// TIA Portal project "lab4" (V15)
// generatory

(* hardware
DEVICE "S7-1200 station_1"  S7-1200 Station
   slot 0: "Rack_0"  S7-1200 Rack  Rack  V1.0
   slot 1: "PLC_1"  CPU 1214C DC/DC/DC  6ES7 214-1AG40-0XB0  V4.2
      slot 3: "AQ 1x12BIT_1"  AQ1 signal board  6ES7 232-4HA30-0XB0  V1.0
   slot 101: "CM 1243-5"  CM 1243-5  6GK7 243-5DX30-0XE0  V1.3
   slot 102: "CM 1241 (RS485)_1"  CM 1241 (RS485)  6ES7 241-1CH30-0XB0  V1.0
*)

// ===== PLC "PLC_1"  CPU 1214C DC/DC/DC =====

VAR_GLOBAL   // PLC tag table "Default tag table"
   "start1" AT %I0.0 : Bool;
   "sprzezenie1" AT %M0.0 : Bool;
   "wyjscie1" AT %Q0.0 : Bool;
   "start2" AT %I0.1 : Bool;
   "sprzezenie2" AT %M0.2 : Bool;
   "WY_1" AT %Q0.2 : Bool;
   "start3" AT %I0.4 : Bool;
   "sprzezenie3" AT %M0.3 : Bool;
   "WY" AT %Q0.3 : Bool;
   "start5" AT %I0.5 : Bool;
   "sprzezenie4" AT %M0.5 : Bool;
   "wyjscie5" AT %Q0.5 : Bool;
   "szpikaZbocze" AT %M1.0 : Bool;
END_VAR

// folder: System blocks/Program resources

DATA_BLOCK "T1"   // DB1
{ S7_Optimized_Access := 'TRUE' }
AUTHOR : Simatic
FAMILY : IEC
NAME : IEC_TMR
VERSION : 1.0
// stored: InstanceOfName IEC_TIMER
"IEC_TIMER"
BEGIN
END_DATA_BLOCK

DATA_BLOCK "t2"   // DB2
{ S7_Optimized_Access := 'TRUE' }
AUTHOR : Simatic
FAMILY : IEC
NAME : IEC_TMR
VERSION : 1.0
// stored: InstanceOfName IEC_TIMER
"IEC_TIMER"
BEGIN
END_DATA_BLOCK

DATA_BLOCK "T3"   // DB3
{ S7_Optimized_Access := 'TRUE' }
AUTHOR : Simatic
FAMILY : IEC
NAME : IEC_TMR
VERSION : 1.0
// stored: InstanceOfName IEC_TIMER
"IEC_TIMER"
BEGIN
END_DATA_BLOCK

DATA_BLOCK "T4"   // DB4
{ S7_Optimized_Access := 'TRUE' }
AUTHOR : Simatic
FAMILY : IEC
NAME : IEC_TMR
VERSION : 1.0
// stored: InstanceOfName IEC_TIMER
"IEC_TIMER"
BEGIN
END_DATA_BLOCK

DATA_BLOCK "T5"   // DB5
{ S7_Optimized_Access := 'TRUE' }
AUTHOR : Simatic
FAMILY : IEC
NAME : IEC_TMR
VERSION : 1.0
// stored: InstanceOfName IEC_TIMER
"IEC_TIMER"
BEGIN
END_DATA_BLOCK

DATA_BLOCK "T6"   // DB6
{ S7_Optimized_Access := 'TRUE' }
AUTHOR : Simatic
FAMILY : IEC
NAME : IEC_TMR
VERSION : 1.0
// stored: InstanceOfName IEC_TIMER
"IEC_TIMER"
BEGIN
END_DATA_BLOCK

DATA_BLOCK "T7"   // DB7
{ S7_Optimized_Access := 'TRUE' }
AUTHOR : Simatic
FAMILY : IEC
NAME : IEC_TMR
VERSION : 1.0
// stored: InstanceOfName IEC_TIMER
"IEC_TIMER"
BEGIN
END_DATA_BLOCK

// folder: (top level)

ORGANIZATION_BLOCK "Main"   // OB1, LAD, ProgramCycle
TITLE = "Main Program Sweep (Cycle)"
{ S7_Optimized_Access := 'TRUE' }
VERSION : 0.1
   VAR_INPUT
      Initial_Call : Bool;   // Initial call of this OB
      Remanence : Bool;   // =True, if remanent data are available
   END_VAR
   VAR_TEMP   // added for the SCL form of the ladder/FBD networks
      _w1 : Bool;
   END_VAR
BEGIN

REGION Network 1: generator szplikowy
   // uzycie do potencjometrow cyfrowych
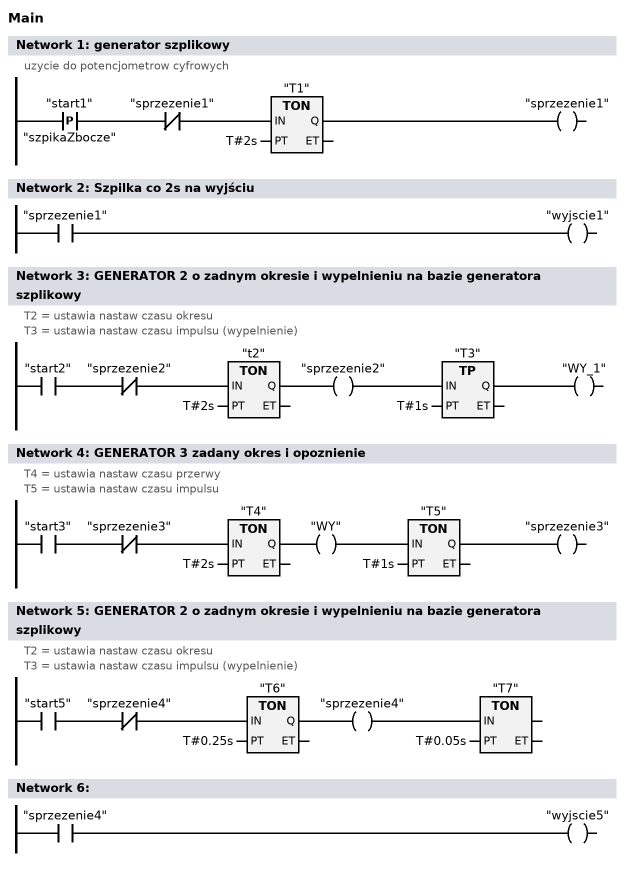
   #_w1 := "start1" AND NOT "szpikaZbocze";   // rising edge of "start1"
   "szpikaZbocze" := "start1";
   "T1".TON(IN := #_w1 AND NOT "sprzezenie1", PT := T#2s);
   "sprzezenie1" := "T1".Q;
END_REGION

REGION Network 2: Szpilka co 2s na wyjściu
   RUNG wire#powerrail
      Contact( "sprzezenie1" )
      Coil( "wyjscie1" )
   END_RUNG
   // the same network as SCL:
   "wyjscie1" := "sprzezenie1";
END_REGION

REGION Network 3: GENERATOR 2 o zadnym okresie i wypelnieniu na bazie generatora szplikowy
   // T2 = ustawia nastaw czasu okresu
   // T3 = ustawia nastaw czasu impulsu (wypelnienie)
   "t2".TON(IN := "start2" AND NOT "sprzezenie2", PT := T#2s);
   "sprzezenie2" := "t2".Q;
   "T3".TP(IN := "t2".Q, PT := T#1s);
   "WY_1" := "T3".Q;
END_REGION

REGION Network 4: GENERATOR 3 zadany okres i opoznienie
   // T4 = ustawia nastaw czasu przerwy
   // T5 = ustawia nastaw czasu impulsu
   "T4".TON(IN := "start3" AND NOT "sprzezenie3", PT := T#2s);
   "WY" := "T4".Q;
   "T5".TON(IN := "T4".Q, PT := T#1s);
   "sprzezenie3" := "T5".Q;
END_REGION

REGION Network 5: GENERATOR 2 o zadnym okresie i wypelnieniu na bazie generatora szplikowy
   // T2 = ustawia nastaw czasu okresu
   // T3 = ustawia nastaw czasu impulsu (wypelnienie)
   "T6".TON(IN := "start5" AND NOT "sprzezenie4", PT := T#0.25s);
   "sprzezenie4" := "T6".Q;
   "T7".TON(IN := "T6".Q, PT := T#0.05s);
END_REGION

REGION Network 6
   RUNG wire#powerrail
      Contact( "sprzezenie4" )
      Coil( "wyjscie5" )
   END_RUNG
   // the same network as SCL:
   "wyjscie5" := "sprzezenie4";
END_REGION
END_ORGANIZATION_BLOCK